FUNCTION TryConvert_UDINT_TO_BOOL : BOOL
VAR_INPUT
	in : UDINT;
	out : REFERENCE TO BOOL;
END_VAR

out := UDINT_TO_BOOL(in);
TryConvert_UDINT_TO_BOOL := TRUE;

END_FUNCTION

(* stored: Version 1.1.0.1, ProductVersion 3.1.4024.12
   POU TryConvert_UDINT_TO_BOOL: Id {1fdc02be-a825-48be-b57c-9822364e7db1}, SpecialFunc None *)
